// TwinCAT 3 PLC project Untitled1
// ProgramVersion: 3.1.4024.0
// libraries:
//   Tc2_Standard, * (Beckhoff Automation GmbH)
//   Tc2_System, * (Beckhoff Automation GmbH)
//   Tc3_Module, * (Beckhoff Automation GmbH)
// project tree:
//   DUTs/ ST_Pompe_Prio.TcDUT
//   FBs/ fb_OrdreAllumage_3.TcPOU, FB_Prio_N.TcPOU, Objet_OrdreAllumage.TcDUT
//   FBs/FB_Temporaire/ FB_LimitationDebit.TcPOU
//   GVLs/ GVL_IO.TcGVL
//   / PlcTask.TcTTO
//   POUs/ MAIN.TcPOU, POU_TEST.TcPOU
// real-time tasks:
//   TASK PlcTask: cycle T#10ms, priority 20, ADS port 350
// I/O:
//   DEVICE Device 1 (EtherCAT) (disabled), AmsNetId 192.168.224.74.2.1
//     Term 1 (EK1200) [EK1200-5000 EtherCAT Power supply (2A E-Bus)]
//       EL1809 1 [EL1809 16Ch. Dig. Input 24V, 3ms]

CONFIGURATION Untitled1
    RESOURCE PLC ON TwinCAT3
        TASK PlcTask(INTERVAL := T#10ms, PRIORITY := 20);
        PROGRAM MAIN WITH PlcTask : MAIN;
    END_RESOURCE
END_CONFIGURATION

// ---- DUTs/ST_Pompe_Prio.TcDUT
TYPE ST_Pompe_Prio :
STRUCT
PmpID				:INT;
Dispox				:BOOL;
PmpPrioNumero		:INT;
Allume				:BOOL;


	

END_STRUCT
END_TYPE

// ---- FBs/Objet_OrdreAllumage.TcDUT
TYPE Objet_OrdreAllumage :
STRUCT
	Numero : INT;
	Disponible : BOOL;
	Allume : BOOL;
END_STRUCT
END_TYPE

// ---- GVLs/GVL_IO.TcGVL
{attribute 'qualified_only'}
VAR_GLOBAL
	
(*

 {attribute 'TcLinkTo' := 'TIID^Device 1 (EtherCAT)^Term 1 (EK1200)^Term 2 (EL1809)^Channel 1^Input'}
 
 TT41_MES AT %I* : BOOL;
 
  {attribute 'TcLinkTo' := 'TIID^Device 1 (EtherCAT)^Term 1 (EK1200)^Term 2 (EL1809)^WcState^WcState'}
 
  WClinkM AT %I* : BOOL;
 
 {attribute 'TcLinkTo' := 'TIID^Device 1 (EtherCAT)^Term 1 (EK1200)^Term 2 (EL1809)^InfoData^State'}
 
  staee AT %Q* : BOOL;
 
  
  *)
  
 //{attribute 'TcLinkTo' := 'TIID^Device 1 (EtherCAT)^Term 1 (EK1200)^Term 2 (EL1809)^InfoData^State'}
   {attribute 'TcLinkTo' := 'TIID^Device 1 (EtherCAT)^Term 1 (EK1200)^EL1809 1^Channel 1^Output'}
 
 TT41_DEFAUT AT %I* : BOOL;

END_VAR




// Term 2 (EL1809)

// ---- POUs/MAIN.TcPOU
PROGRAM MAIN

VAR	

PRIO_P	:FB_Prio_N;

PrioActuel:	STRING;

TestPrioFB: fb_OrdreAllumage_3;
	object: ARRAY [1..3] OF Objet_OrdreAllumage;
	nbrobjallume: INT;
	ordrprio: STRING;
	optiordraluu: BOOL;
	nbrobjallumee: INT;
	prioactu: STRING;
	errorr: BOOL;
	serror: STRING;
	
	LimitationDebit: FB_LimitationDebit;

	bCmdOn: BOOL;
	bDefautFIT1: BOOL;
	bDefautFIT2: BOOL;
	rMesureFIT2: REAL;
	rSeuilDebit: REAL;
	tTempsActivation: TIME;
	rVitessePompe1: REAL;
	rVitessePompe2: REAL;
	rVitessePompe3: REAL;
	rVitessePompe4: REAL;
	bStatusOn: BOOL;
	rVitesseLimPompe1: REAL;
	rVitesseLimPompe2: REAL;
	rVitesseLimPompe3: REAL;
	rVitesseLimPompe4: REAL;
	rMesureFIT1: REAL;
	testt: UINT;
END_VAR




VAR CONSTANT
	
END_VAR

PRIO_P(
	Prio_P:=PrioActuel);
TestPrioFB(
	Objet:= object, 
	iNbreObjet_A_Allumer:=nbrobjallume , 
	sOrdreDePriorite:=ordrprio , 
	bOptimisationOrdreAllumage:=optiordraluu , 
	iNbreObjetAllume=>nbrobjallumee , 
	sPrioriteActuelle=> prioactu, 
	bError=> errorr, 
	sError=> serror);


testt:=1+1;

	
LimitationDebit(
	bCmdOn:= bCmdOn , 
	bDefautFIT1:= bDefautFIT1, 
	bDefautFIT2:= bDefautFIT2, 
	rMesureFIT1:= rMesureFIT1 , 
	rMesureFIT2:= rMesureFIT2 , 
	rSeuilDebit:= rSeuilDebit, 
	tTempsActivation:= tTempsActivation , 
	rVitessePompe1:= rVitessePompe1 , 
	rVitessePompe2:= rVitessePompe2 , 
	rVitessePompe3:= rVitessePompe3, 
	rVitessePompe4:= rVitessePompe4, 
	bStatusOn=> bStatusOn , 
	rVitesseLimPompe1=> rVitesseLimPompe1, 
	rVitesseLimPompe2=> rVitesseLimPompe2, 
	rVitesseLimPompe3=> rVitesseLimPompe3, 
	rVitesseLimPompe4=> rVitesseLimPompe4);

	
rVitessePompe1:=rVitessePompe2:=rVitessePompe3:=rVitessePompe4:=rVitessePompe1+ 0.0001;

END_PROGRAM

// ---- FBs/FB_Prio_N.TcPOU
FUNCTION_BLOCK FB_Prio_N
VAR_INPUT
Prio_P	:STRING;
DispoPmp1	:BOOL;
DispoPmp2	:BOOL;
DispoPmp3	:BOOL;
DispoPmp4	:BOOL;
Tab_PrioPomp: ARRAY [1..4] OF STRING;
 
END_VAR
VAR_OUTPUT
	Priorite_PompeOut	:STRING; 
END_VAR
VAR
	
Tab_Pompe_Prio_IN	:ARRAY[1..4] OF ST_Pompe_Prio;
Tab_Pompe_Prio_Temp	:ARRAY[1..4] OF ST_Pompe_Prio;
Tab_Pompe_Prio_OUT	:ARRAY[1..4] OF ST_Pompe_Prio;
i	:INT;
j	:INT;
Tab_Temp	:ST_Pompe_Prio;
	PompeDispo: INT;
	Tab_Pompe_Prio_TempdisP :ARRAY[1..4] OF ST_Pompe_Prio;
	Arret: INT;
	PmpDispo: INT;
	x: INT;
	PrioritePompe: STRING(INT#4);
END_VAR

 
// affectation de la priorité des pompes a chaque pompes 
FOR i:=1 TO 4 BY 1 DO
	
	Tab_Pompe_Prio_IN[I].PmpID:= STRING_TO_INT (MID (Prio_P,1,i));
	Tab_Pompe_Prio_IN[I].PmpPrioNumero:=i;
	             	
END_FOR

// affectation des dispo aux pompes


FOR j:=1 TO 4 BY 1 DO
	
	IF Tab_Pompe_Prio_IN[j].PmpID=1 THEN 
		Tab_Pompe_Prio_IN[j].Dispox:=DispoPmp1;
	ELSIF Tab_Pompe_Prio_IN[j].PmpID=2 THEN 
		Tab_Pompe_Prio_IN[j].Dispox:=DispoPmp2;
	ELSIF Tab_Pompe_Prio_IN[j].PmpID=3 THEN 
		Tab_Pompe_Prio_IN[j].Dispox:=DispoPmp3;
	ELSIF Tab_Pompe_Prio_IN[j].PmpID=4 THEN 
		Tab_Pompe_Prio_IN[j].Dispox:=DispoPmp4;	
	END_IF
END_FOR 

Tab_Pompe_Prio_IN[1].PmpID;
              
Tab_Pompe_Prio_IN[2].PmpID;
              
Tab_Pompe_Prio_IN[3].PmpID;
             
Tab_Pompe_Prio_IN[4].PmpID;

 // affecter les pompes disponibles dans un tableau pour savoir combien de pmp dispo
j:=1;
i:=1;
x:=0;

FOR i:=1 TO 4 BY 1 DO
	IF 	Tab_Pompe_Prio_IN[i].Dispox=TRUE THEN
		Tab_Pompe_Prio_Tempdisp[j]:=Tab_Pompe_Prio_IN[i];
		j:=j+1;
	ELSE
		Tab_Pompe_Prio_Tempdisp[4-X].PmpID:=0;
		x:=x+1;
	END_IF
	
	PmpDispo:=j-1;
END_FOR

Tab_PrioPomp[1]:= INT_TO_STRING(Tab_Pompe_Prio_Tempdisp[1].PmpID);
Tab_PrioPomp[2]:= INT_TO_STRING(Tab_Pompe_Prio_Tempdisp[2].PmpID);
Tab_PrioPomp[3]:= INT_TO_STRING(Tab_Pompe_Prio_Tempdisp[3].PmpID);
Tab_PrioPomp[4]:= INT_TO_STRING(Tab_Pompe_Prio_Tempdisp[4].PmpID);



IF  0 < pmpdispo AND pmpdispo <5 THEN
	
	Priorite_PompeOut:='';	
	FOR i:=1 TO pmpdispo BY 1 DO 
		
		Priorite_PompeOut:=concat (Priorite_PompeOut, Tab_PrioPomp[i]);
	
	END_FOR	
ELSE 	Priorite_PompeOut:='0	';
END_IF	


(* code pour tri ordre croissant
FOR i:=1 TO 3 BY 1 DO
	
	FOR j:=1 TO 4 - i BY 1 DO
		IF 		Tab_Pompe_Prio_temp[i].PmpID >= Tab_Pompe_Prio_Temp[j+1].PmpID THEN
			
			Tab_Temp:=Tab_Pompe_Prio_Temp[j];
			Tab_Pompe_Prio_Temp[j]:=Tab_Pompe_Prio_Temp[j+1];
			Tab_Pompe_Prio_Temp[j+1]:=Tab_Temp;
		END_IF
	END_FOR
	
END_FOR
*)

END_FUNCTION_BLOCK

// ---- FBs/fb_OrdreAllumage_3.TcPOU
FUNCTION_BLOCK fb_OrdreAllumage_3
VAR_IN_OUT
	Objet : ARRAY[1..iNbreObjet] OF Objet_OrdreAllumage; //Tableau d'objet que l'on souhaite allumer (à renseigner dans l'ordre croissant)
END_VAR
VAR_INPUT	
	iNbreObjet_A_Allumer : INT; //Nombre d'objet qui ont besoin d'etre allumé
	sOrdreDePriorite : STRING; //Inscrire ici l'ordre de priorité ex : 123
	bOptimisationOrdreAllumage : BOOL := TRUE; //Indique si on souhaite conserver un objet déja en fonctionnement alors qu'un objet de priorité plus grande devient disponible
END_VAR
VAR_OUTPUT
	iNbreObjetAllume : INT; //Nombre d'objet allumé
	sPrioriteActuelle : STRING;
	bError : BOOL;
	sError : STRING;
END_VAR
VAR
	i : INT;
	j : INT;
	iCaseTri : INT;
	iIndexPointeurPriorite : INT;
	iNbreObjetRestant_A_Allumer : INT;
	iNbreObjetNonDispo : INT;
	iTailleOrdrePriorite : INT;
	ObjetTrie : ARRAY[1..iNbreObjet] OF Objet_OrdreAllumage; //Tableau trié par priorité
	aPrioriteActuelle : ARRAY[1..iNbreObjet] OF INT;
END_VAR
VAR CONSTANT
	iNbreObjet : INT := 3; //Renseigner ici le nombre d'objet
END_VAR

(* Ce fb permet d'allumer des objets dans l'ordre de priorité du tableau.
 Si un objet est déja allumé, alors meme si il n'est pas le plus prioritaire, il reste allumé et garde la priorité jusqu'a ce qu'il soit éteint.
 Une fois éteint, si on le remet dans son bon ordre de priorité*)
 
 //Tri du tableau en fonction de la priorité demandée et gestion d'erreur
 iTailleOrdrePriorite := LEN(sOrdreDePriorite);
IF iTailleOrdrePriorite <> iNbreObjet THEN //Si l'ordre de priorité ne correspond pas au nombre d'objet, il y a une erreur
	bError := TRUE;
	sError := 'l$'ordre de priorité ne correspond pas au nombre d$'objet';
	RETURN; 
END_IF

FOR i := 1 TO iNbreObjet DO //On tri en fonction de la priorité
	iCaseTri := STRING_TO_INT(MID(sOrdreDePriorite, 1, i));
	IF iCaseTri > iNbreObjet THEN
		bError := TRUE;
		sError := 'Il y a un ordre de priorité plus grand que le nombre d$'objets';
		RETURN; 
	ELSE
		ObjetTrie[i] := Objet[iCaseTri];
	END_IF	
END_FOR

FOR i := 1 TO iNbreObjet DO //On regarde si il n'y a pas deux fois le meme objet dans la priorité
	FOR j := 1 TO iNbreObjet DO
		IF i <> j AND ObjetTrie[i].Numero = ObjetTrie[j].Numero THEN
			bError := TRUE;
			sError := 'Il y a plusieurs fois le meme objet dans l$'ordre de priorité';
			RETURN; 
		END_IF
	END_FOR
END_FOR

//Si on va jusqu'ici (si on ne va pas dans RETURN), on efface les erreurs
bError := FALSE;
sError := '';



IF bOptimisationOrdreAllumage THEN //Si on souhaite conserver un objet déja en fonctionnement alors qu'un objet de priorité plus grande devient disponible
	//Calcul du nombre d'objet restant à allumer
	iNbreObjetRestant_A_Allumer := iNbreObjet_A_Allumer - iNbreObjetAllume;
	IF iNbreObjetRestant_A_Allumer > 0 THEN  //Allumage des objet disponible
		FOR i := 1 TO iNbreObjet DO
			IF ObjetTrie[i].Disponible  //Si dispo
			 AND NOT ObjetTrie[i].Allume //Si pas déja allumé
			 AND iNbreObjetRestant_A_Allumer > 0 THEN //Si on doit en allumer encore
				ObjetTrie[i].Allume := TRUE; //On allumer
				iNbreObjetRestant_A_Allumer := iNbreObjetRestant_A_Allumer - 1; //On décrémente le nombre d'objets à allumer
			END_IF	 
		END_FOR
	ELSIF iNbreObjetRestant_A_Allumer < 0 THEN //Arret des objets
		FOR i := iNbreObjet TO 1 BY -1 DO
			IF ObjetTrie[i].Allume  //Si allumé
			 AND iNbreObjetRestant_A_Allumer < 0 THEN //Si on doit en éteindre encore
				ObjetTrie[i].Allume := FALSE; //On éteint
				iNbreObjetRestant_A_Allumer := iNbreObjetRestant_A_Allumer + 1; //On incrémente le nombre d'objets à allumer
			END_IF	 
		END_FOR
	END_IF
ELSE //Si on souhaite toujours allumer les objets les plus prioritaires
	iNbreObjetRestant_A_Allumer := iNbreObjet_A_Allumer;
	FOR i := 1 TO iNbreObjet DO
		IF ObjetTrie[i].Disponible  //Si dispo
		 AND iNbreObjetRestant_A_Allumer > 0 THEN //Si on doit en allumer encore
			ObjetTrie[i].Allume := TRUE; //On allumer
			iNbreObjetRestant_A_Allumer := iNbreObjetRestant_A_Allumer - 1; //On décrémente le nombre d'objets à allumer
		ELSIF iNbreObjetRestant_A_Allumer = 0 THEN //Si on ne doit plus en allumer
			ObjetTrie[i].Allume := FALSE; //On éteint les autres
		END_IF			
	END_FOR
END_IF


 //Calcul du nombre d'objet allumé. On éteint les objet non disponible. 
 iNbreObjetAllume := 0;
 iNbreObjetNonDispo := 0;
FOR i := 1 TO iNbreObjet DO
	IF ObjetTrie[i].Allume AND ObjetTrie[i].Disponible THEN
		iNbreObjetAllume := iNbreObjetAllume + 1;
	ELSIF ObjetTrie[i].Allume AND NOT ObjetTrie[i].Disponible THEN
		ObjetTrie[i].Allume := FALSE;
	END_IF
	IF NOT ObjetTrie[i].Disponible THEN //On calcul le nombre d'objets non disponible
		iNbreObjetNonDispo := iNbreObjetNonDispo + 1;
	END_IF
END_FOR
 
 //On reseigne l'ordre de priorité actuel (en fonction des disponibilité et des objets déja allumé)
iIndexPointeurPriorite := 1;
IF iNbreObjetAllume > 0 THEN //On cherche dans un premier temps les objets dispo et allumée
	FOR i := 1 TO iNbreObjet DO 
		IF ObjetTrie[i].Disponible AND ObjetTrie[i].Allume THEN
			aPrioriteActuelle[iIndexPointeurPriorite] := ObjetTrie[i].Numero; 
			iIndexPointeurPriorite := iIndexPointeurPriorite + 1;
		END_IF
	END_FOR
END_IF

FOR i := 1 TO iNbreObjet DO  //On met ensuite selon la dispo
	IF ObjetTrie[i].Disponible AND NOT ObjetTrie[i].Allume THEN
		aPrioriteActuelle[iIndexPointeurPriorite] := ObjetTrie[i].Numero; 
		iIndexPointeurPriorite := iIndexPointeurPriorite + 1;
	END_IF
END_FOR

//On met la priorité actuelle dans un STRING
sPrioriteActuelle := '';
FOR i := 1 TO iNbreObjet - iNbreObjetNonDispo DO 
	sPrioriteActuelle := CONCAT(sPrioriteActuelle, INT_TO_STRING(aPrioriteActuelle[i]));
END_FOR


  //On remet les paramètres du tableau trié dans le tableau rangé en ordre croissant
FOR i := 1 TO iNbreObjet DO
	FOR j := 1 TO iNbreObjet DO
		IF Objet[i].Numero = ObjetTrie[j].Numero THEN
			Objet[i] := ObjetTrie[j];
		END_IF	 
	END_FOR
END_FOR

END_FUNCTION_BLOCK

// ---- FBs/FB_Temporaire/FB_LimitationDebit.TcPOU
FUNCTION_BLOCK FB_LimitationDebit
VAR_INPUT
	bCmdOn			:BOOL:= FALSE; 	//Commande de démarrage de la fonction (désactivée par défaut)
	bDefautFIT1		:BOOL;		// Defaut capteur débit 1
 	bDefautFIT2		:BOOL;		// Defaut capteur débit 2
	rMesureFIT1		:REAL;		// Mzsure capteur débit 1
	rMesureFIT2		:REAL;		// Mzsure capteur débit 2
	rSeuilDebit 	:REAL; 		// Seuil debit a ne pas depasser >> renseigner par operateur
	tTempsActivation:TIME;		// tempo pour activer la fonction 
	rVitessePompe1	:REAL;		// Vitesse Pompe1	>> connecter avec la consigne de vitesse de la pompe 1
	rVitessePompe2	:REAL;		// Vitesse Pompe2	>> connecter avec la consigne de vitesse de la pompe 2
	rVitessePompe3	:REAL;		// Vitesse Pompe3	>> connecter avec la consigne de vitesse de la pompe 3
	rVitessePompe4	:REAL;		// Vitesse Pompe4	>> connecter avec la consigne de vitesse de la pompe 4
END_VAR


VAR_OUTPUT
	bStatusOn		: BOOL; //Retour d'état du fonctionnement de la fonction 
	rVitesseLimPompe1	:REAL;		// Vitesse Pompe1	>> connecter avec la consigne de vitesse de la pompe 1
	rVitesseLimPompe2	:REAL;		// Vitesse Pompe2	>> connecter avec la consigne de vitesse de la pompe 2
	rVitesseLimPompe3	:REAL;		// Vitesse Pompe3	>> connecter avec la consigne de vitesse de la pompe 3
	rVitesseLimPompe4	:REAL;		// Vitesse Pompe4	>> connecter avec la consigne de vitesse de la pompe 4

END_VAR


VAR
	tTempoSEUILDEBITPDIC41001		:TON;		// tempo demarrage arret fonction limitation debit rcu retour reseau
	R_TrigSeuilDebit				:R_TRIG;	// detection de front montant de dépassement seuil debit fonction limitation de debit  
	
END_VAR


// Fonction limitation de débit

IF bCmdOn THEN   // si fonction activéé
	
	IF NOT bDefautFIT1 AND NOT bDefautFIT2 THEN  // si pas de defaut sur les deux capteurs de débit retour réseau général 
		
		IF rSeuilDebit > (rMesureFIT1 + rMesureFIT2) THEN		// si le seuil de débit est superieur au débit général retour RCU 
			tTempoSEUILDEBITPDIC41001(IN:=TRUE,PT:=tTempsActivation);	// tempo avant d'activer la fonction
			IF tTempoSEUILDEBITPDIC41001.Q THEN
				bStatusOn:=TRUE; 	// Status ON de la fonction
				tTempoSEUILDEBITPDIC41001(IN:=FALSE);
				R_TrigSeuilDebit(CLK:=bStatusOn);
			END_IF
			
			IF R_TrigSeuilDebit.Q THEN	// sauvegardé les consignes de vitesse des pompes
				rVitesseLimPompe1:=rVitessePompe1; 
				rVitesseLimPompe2:=rVitessePompe2; 
				rVitesseLimPompe3:=rVitessePompe3; 
				rVitesseLimPompe4:=rVitessePompe4;
			END_IF
		ELSE
			bStatusOn:=FALSE; 	// Status OFF de la fonction 	
			tTempoSEUILDEBITPDIC41001(IN:=FALSE);					// INIT la tempo
			R_TrigSeuilDebit(CLK:=bStatusOn);
		END_IF
		
	ELSE
	bStatusOn:=FALSE; 	// Status OFF de la fonction 	
	tTempoSEUILDEBITPDIC41001(IN:=FALSE);					// INIT la tempo
	R_TrigSeuilDebit(CLK:=bStatusOn);
	END_IF
ELSE
	bStatusOn:=FALSE;  	// Status OFF de la fonction
	tTempoSEUILDEBITPDIC41001(IN:=FALSE);					// INIT la tempo
	R_TrigSeuilDebit(CLK:=bStatusOn);
END_IF



(*
// SI consigne vitesse PID est < a la rVitesseLimPompe et fonction limitation debit actif alors on prend la vitesse du PID 
IF bCmdOn AND bStatusOn THEN
	IF RM pompe1 THEN 
		IF  rVitesseLimPompe1> rVitessePompe1 THEN 
			
		rVitesseLimPompe1:=rVitessePompe1;	
		rVitesseLimPompe2:=rVitessePompe2;
		rVitesseLimPompe3:=rVitessePompe3;
		
		END_IF
	END_IF
END_IF
*)

END_FUNCTION_BLOCK

// ---- POUs/POU_TEST.TcPOU
PROGRAM POU_TEST
VAR
	
TEST	:fb_OrdreAllumage_3; 
END_VAR

TEST(
	Objet:= , 
	iNbreObjet_A_Allumer:= , 
	sOrdreDePriorite:= , 
	bOptimisationOrdreAllumage:= , 
	iNbreObjetAllume=> , 
	sPrioriteActuelle=> , 
	bError=> , 
	sError=> );

END_PROGRAM
